FUNCTION_BLOCK FB_NciChannelTangential EXTENDS FB_ComponentBase IMPLEMENTS I_NciChannel_FeedTable

VAR_INPUT
    stAxisIds : ST_NciAxisIds;
	nGroupId  : UDINT := 5;
END_VAR

VAR
    stNciToPlc AT %I* : NCTOPLC_NCICHANNEL_REF;
    stPlcToNci AT %Q* : PLCTONC_NCICHANNEL_REF;
	
    // ZMIANA: Blok Ext3DGroup pozwala dodać osie Q1..Q5
    fbBuildExtGroup : CfgBuildExt3DGroup;
    fbUngroup       : CfgReconfigGroup;
    
    // Obsługa Resetu / Start / Stop
    fbStartStop     : ItpStartStopEx;
    fbReset         : ItpResetEx2;

    // --- NOWOŚĆ: Blok do przesyłania tabel z RAMu ---
    fbFeedTable     : FB_NciFeedTable;
    refFeedTable    : REFERENCE TO ST_NciFeedGroupTable; // Przechowuje wskaźnik do tabeli z Executora
    _bExecuteFeed   : BOOL;
    _IsFeedingDone  : BOOL;
    _IsChannelDone  : BOOL;

    _IsGrouped      : BOOL;
    _IsReady		: BOOL;
	
	_bResetFeed : BOOL;
END_VAR

METHOD BuildGroup
_IsGrouped := FALSE;
_Error := FALSE; 
_ErrorId := 0;

fbBuildExtGroup(
    bExecute := TRUE,
    nGroupId := nGroupId,
    nXAxisId := stAxisIds.nX,
    nYAxisId := stAxisIds.nY,
    nZAxisId := stAxisIds.nZ,
    nQ1AxisId := stAxisIds.nQ1 
);
END_METHOD

PROPERTY ChannelError : BOOL
GET
ChannelError := _Error OR (stNciToPlc.ErrorCode <> 0);
END_GET
END_PROPERTY

PROPERTY ChannelErrorId : UDINT
GET
IF stNciToPlc.ErrorCode <> 0 THEN
    ChannelErrorId := stNciToPlc.ErrorCode;
ELSE
    ChannelErrorId := _ErrorId;
END_IF
END_GET
END_PROPERTY

METHOD PUBLIC CyclicLogic
SUPER^.CyclicLogic();


stPlcToNci.ChnAxesOvr := 1000000;


fbBuildExtGroup(tTimeOut := T#2S);
fbUngroup(tTimeOut := T#2S);
fbStartStop(sNciToPlc := stNciToPlc, tTimeOut := T#2S);
fbReset(sNciToPlc := stNciToPlc, tTimeOut := T#2S);


IF __ISVALIDREF(refFeedTable) THEN
    fbFeedTable(
        bExecute := _bExecuteFeed,
        bReset := _bResetFeed,
        stFeedGroupTable := refFeedTable,
        stNciToPlc := stNciToPlc,
        bFeedingDone => _IsFeedingDone,
        bChannelDone => _IsChannelDone
    );
    
 
    IF _bResetFeed THEN
        _bResetFeed := FALSE;
    END_IF


    IF _IsChannelDone OR fbFeedTable.bError THEN
        IF _bExecuteFeed AND _IsChannelDone THEN
            ADSLOGSTR(ADSLOG_MSGTYPE_HINT, 'NciChannelTan: Ruch interpolowany zakonczony (Channel Done).', '');
        END_IF
        _bExecuteFeed := FALSE;
    END_IF
    
    IF fbFeedTable.bError THEN
        IF NOT _Error THEN
            ADSLOGDINT(ADSLOG_MSGTYPE_ERROR, 'NciChannelTan: BLAD FeedTable! Kod: %d', UDINT_TO_DINT(fbFeedTable.nErrorId));
        END_IF
        _Error := TRUE;
        _ErrorId := fbFeedTable.nErrorId;
    END_IF
END_IF


IF fbStartStop.bErr THEN
    IF NOT _Error THEN
        ADSLOGDINT(ADSLOG_MSGTYPE_ERROR, 'NciChannelTan: BLAD StartStop! Kod: %d', UDINT_TO_DINT(fbStartStop.nErrId));
    END_IF
    _Error := TRUE;
    _ErrorId := fbStartStop.nErrId;
    fbStartStop(bStart := FALSE, bStop := FALSE, sNciToPlc := stNciToPlc);
ELSIF fbStartStop.bBusy THEN
    fbStartStop(bStart := FALSE, sNciToPlc := stNciToPlc);
ELSIF NOT fbStartStop.bBusy AND fbStartStop.bStop THEN
    fbStartStop(bStop := FALSE, sNciToPlc := stNciToPlc);
END_IF


IF fbUngroup.bErr THEN
    IF fbUngroup.bExecute THEN
        ADSLOGDINT(ADSLOG_MSGTYPE_ERROR, 'NciChannelTan: BLAD rozpinania grupy! Kod: %d', UDINT_TO_DINT(fbUngroup.nErrId));
    END_IF
    _Error := TRUE;
    _ErrorId := fbUngroup.nErrId;
    fbUngroup(bExecute := FALSE);
    _IsGrouped := FALSE;
ELSIF fbUngroup.bBusy = FALSE AND fbUngroup.bExecute THEN
    ADSLOGSTR(ADSLOG_MSGTYPE_HINT, 'NciChannelTan: Grupa rozpieta pomyslnie.', '');
    _IsGrouped := FALSE;
    fbUngroup(bExecute := FALSE);
END_IF

IF fbBuildExtGroup.bErr THEN
    IF fbBuildExtGroup.bExecute THEN
        ADSLOGDINT(ADSLOG_MSGTYPE_ERROR, 'NciChannelTan: BLAD budowania grupy rozszerzonej! Kod: %d', UDINT_TO_DINT(fbBuildExtGroup.nErrId));
    END_IF
    _Error := TRUE;
    _ErrorId := fbBuildExtGroup.nErrId;
    fbBuildExtGroup(bExecute := FALSE); 
ELSIF fbBuildExtGroup.bBusy = FALSE AND fbBuildExtGroup.bExecute THEN
    ADSLOGSTR(ADSLOG_MSGTYPE_HINT, 'NciChannelTan: Grupa rozszerzona (X,Y,Z,Q) zbudowana pomyslnie.', '');
    _IsGrouped := TRUE;
    fbBuildExtGroup(bExecute := FALSE);
END_IF

IF fbReset.bErr THEN
    _Error := TRUE;
    _ErrorId := fbReset.nErrId;
    fbReset(bExecute := FALSE, sNciToPlc := stNciToPlc);
ELSIF fbReset.bBusy = FALSE AND fbReset.bExecute THEN
    fbReset(bExecute := FALSE, sNciToPlc := stNciToPlc);
END_IF
END_METHOD

PROPERTY IsChannelDone : BOOL
GET
IsChannelDone := _IsChannelDone;
END_GET
END_PROPERTY

PROPERTY IsFeedingDone : BOOL
GET
IsFeedingDone := _IsFeedingDone;
END_GET
END_PROPERTY

PROPERTY IsGrouped : BOOL
GET
IsGrouped := _IsGrouped;
END_GET
END_PROPERTY

PROPERTY IsReady : BOOL
GET
IsReady := (stNciToPlc.ItpState = 2);
END_GET
END_PROPERTY

METHOD ResetChannel
fbStartStop(bStart := FALSE, bStop := FALSE, sNciToPlc := stNciToPlc);

_bResetFeed := TRUE; // <-- ZMIANA: Zamiast lokalnego wywołania, ustawiamy flagę
_bExecuteFeed := FALSE; 

fbReset(
    bExecute := TRUE,
    sNciToPlc := stNciToPlc
);

_Error := FALSE;
_ErrorId := 0;
END_METHOD

METHOD Start
fbStartStop(
    bStart := TRUE, 
    bStop := FALSE,
    sNciToPlc := stNciToPlc 
);
END_METHOD

METHOD StartFeedTable
VAR_IN_OUT
    stTable : ST_NciFeedGroupTable;
END_VAR
// Pobieramy referencję do tabeli (która np. fizycznie leży w Executorze)
refFeedTable REF= stTable;

// Zerujemy flagi gotowości
_IsFeedingDone := FALSE;
_IsChannelDone := FALSE;

// Wyzwalamy blok feedujący
_bExecuteFeed := TRUE;
END_METHOD

METHOD Stop
fbStartStop(
    bStart := FALSE, 
    bStop := TRUE,
    sNciToPlc := stNciToPlc
);
END_METHOD

METHOD Ungroup
fbUngroup(
    bExecute := TRUE, 
    nGroupId := nGroupId
);
END_METHOD

END_FUNCTION_BLOCK

(* stored: Version 1.1.0.1, ProductVersion 3.1.4024.15
   POU FB_NciChannelTangential: Id {e0b2b8c9-715d-4f01-9a7c-12345678abcd}, SpecialFunc None
   Method BuildGroup: Id {c51e0640-5bb9-4b6a-9a99-b1411b933d1c}
   Property ChannelError: Id {1584ea0b-bc17-48f8-b7eb-d4cfd96c92d5}
   Get Get: Id {f5d21a52-b886-4f4f-b673-d56b6a070eb3}
   Property ChannelErrorId: Id {f3d3283f-df3d-4cba-a15d-85ad21c97a55}
   Get Get: Id {6263884b-dfa8-4c28-bb7e-f55bc8120468}
   Method CyclicLogic: Id {45df0f02-a1b4-4bca-86ff-90a8a65b06a0}
   Property IsChannelDone: Id {b2c3d4e5-f6a7-5890-1234-bcdef0123456}
   Get Get: Id {f5d21a52-b886-4f4f-b673-d56b6a070e23}
   Property IsFeedingDone: Id {a1b2c3d4-e5f6-4789-0123-abcdef123456}
   Get Get: Id {f5d21a52-b886-4f4f-b673-d56b6a070e12}
   Property IsGrouped: Id {ca4a1db1-b5fb-419b-ab09-72f5342a3922}
   Get Get: Id {62b55f11-ffc5-43ea-98fb-7cfbcbf4d26b}
   Property IsReady: Id {8cb00010-cfbd-4bc9-bb17-8e1041b3a5ef}
   Get Get: Id {e146eb11-6677-4952-acc3-dbdd922bf07d}
   Method ResetChannel: Id {dc04c0d4-1a98-4c91-a18d-f5e02a11b655}
   Method Start: Id {cd971ad7-0452-49be-824a-feb5ae9fdcf4}
   Method StartFeedTable: Id {e1f2f3f4-5a6b-7c8d-9e0f-1a2b3c4d5e6f}
   Method Stop: Id {3a0bc19e-e373-45ab-a70e-e479a419ebf4}
   Method Ungroup: Id {6ad59f51-b0db-424f-ba3b-01fc63478ab8} *)
